// TIA Portal V16 export
// export: Created 2022-05-05T19:56:47.8854088Z, ExportSetting WithDefaults, DisplayName Totally Integrated Automation Portal, DisplayVersion V16 Update 2, DisplayName TIA Portal Version Control Interface, DisplayVersion V16 Update 2, DisplayName TIA Portal Openness, DisplayVersion V16 Update 2, DisplayName SINAMICS Startdrive Advanced, DisplayVersion V16 Update 5, DisplayName SINAMICS Startdrive G130, G150, S120, S150, SINAMICS MV, S210, DisplayVersion V16 Update 5, DisplayName SINAMICS Startdrive G110M, G120, G120C, G120D, G120P, G115D, DisplayVersion V16 Update 5, DisplayName STEP 7 Professional, DisplayVersion V16 Update 2, DisplayName SIMATIC Energy Suite, DisplayVersion V16, DisplayName STEP 7 Safety, DisplayVersion V16, DisplayName SINUMERIK 840D sl STEP 7 Toolbox, DisplayVersion V16, DisplayName Simocode ES, DisplayVersion V16, DisplayName WinCC Professional, DisplayVersion V16 Update 2, DisplayName SIMATIC Visualization Architect, DisplayVersion V16
ORGANIZATION_BLOCK "Main"   // OB1, LAD, ProgramCycle
TITLE = "Main Program Sweep (Cycle)"
{ S7_Optimized_Access := 'TRUE' }
VERSION : 0.1
// stored: AutoNumber true, IsIECCheckEnabled false, SetENOAutomatically false
   VAR_INPUT
      Initial_Call : Bool;   // Initial call of this OB
      Remanence : Bool;   // =True, if remanent data are available
   END_VAR
   VAR_TEMP   // added for the SCL form of the ladder/FBD networks
      _w1 : Bool;
      _w2 : Bool;
      _w3 : Bool;
      _w4 : Bool;
   END_VAR
BEGIN

REGION Network 1: Reset
   // Detect when Factory I/O starts running, reset state
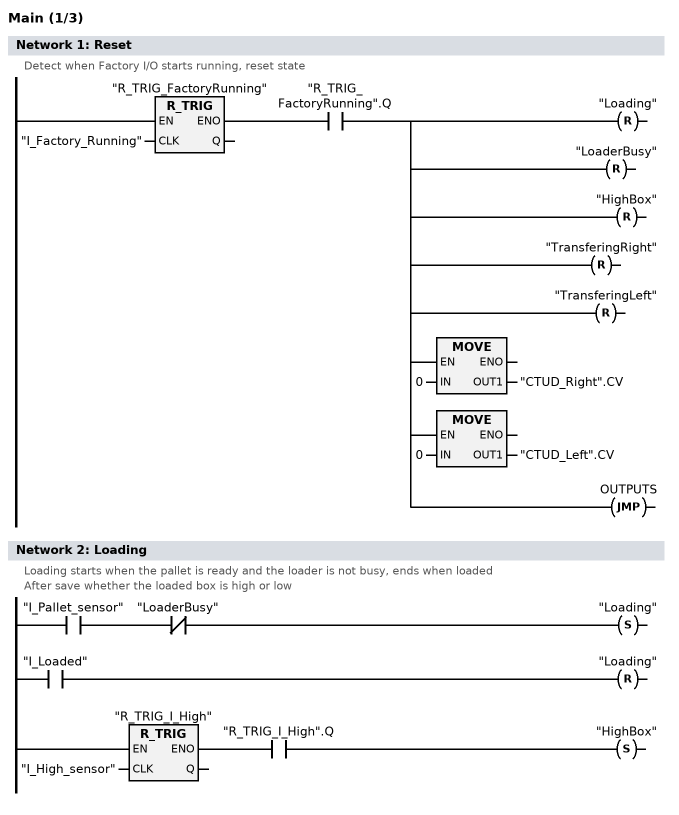
   RUNG wire#powerrail
      "R_TRIG_FactoryRunning".R_TRIG(CLK := "I_Factory_Running", Q =>)
      Contact( "R_TRIG_FactoryRunning".Q )
      wire#w1
      R_Coil( "Loading" )
   END_RUNG
   RUNG wire#w1
      R_Coil( "LoaderBusy" )
   END_RUNG
   RUNG wire#w1
      R_Coil( "HighBox" )
   END_RUNG
   RUNG wire#w1
      R_Coil( "TransferingRight" )
   END_RUNG
   RUNG wire#w1
      R_Coil( "TransferingLeft" )
   END_RUNG
   RUNG wire#w1
      Move(in := 0, out1 => "CTUD_Right".CV)
   END_RUNG
   RUNG wire#w1
      Move(in := 0, out1 => "CTUD_Left".CV)
   END_RUNG
   RUNG wire#w1
      JumpCoil( OUTPUTS )
   END_RUNG
   // the same network as SCL:
   "R_TRIG_FactoryRunning"(CLK := "I_Factory_Running", ENO => #_w1);   // R_TRIG
   #_w2 := #_w1 AND "R_TRIG_FactoryRunning".Q;
   IF #_w2 THEN
       "Loading" := FALSE;
       "LoaderBusy" := FALSE;
       "HighBox" := FALSE;
       "TransferingRight" := FALSE;
       "TransferingLeft" := FALSE;
       "CTUD_Right".CV := 0;
       "CTUD_Left".CV := 0;
       GOTO OUTPUTS;
   END_IF;
END_REGION

REGION Network 2: Loading
   // Loading starts when the pallet is ready and the loader is not busy, ends when loaded
   // After save whether the loaded box is high or low
   RUNG wire#powerrail
      Contact( "I_Pallet_sensor" )
      I_Contact( "LoaderBusy" )
      S_Coil( "Loading" )
   END_RUNG
   RUNG wire#powerrail
      Contact( "I_Loaded" )
      R_Coil( "Loading" )
   END_RUNG
   RUNG wire#powerrail
      "R_TRIG_I_High".R_TRIG(CLK := "I_High_sensor", Q =>)
      Contact( "R_TRIG_I_High".Q )
      S_Coil( "HighBox" )
   END_RUNG
   // the same network as SCL:
   IF "I_Pallet_sensor" AND NOT "LoaderBusy" THEN "Loading" := TRUE; END_IF;
   IF "I_Loaded" THEN "Loading" := FALSE; END_IF;
   "R_TRIG_I_High"(CLK := "I_High_sensor", ENO => #_w1);   // R_TRIG
   IF #_w1 AND "R_TRIG_I_High".Q THEN "HighBox" := TRUE; END_IF;
END_REGION

REGION Network 3: Transfer
   // Decide where to transfer after loading
   // Loader busy if loading or transfering
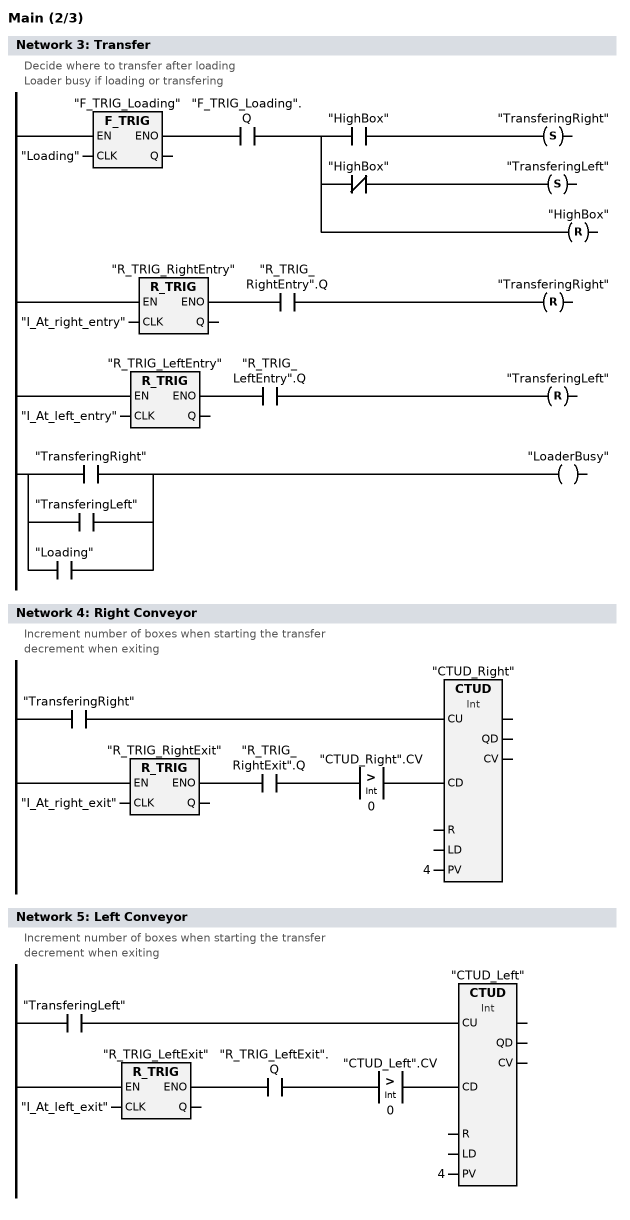
   RUNG wire#powerrail
      "F_TRIG_Loading".F_TRIG(CLK := "Loading", Q =>)
      Contact( "F_TRIG_Loading".Q )
      wire#w1
      Contact( "HighBox" )
      S_Coil( "TransferingRight" )
   END_RUNG
   RUNG wire#w1
      I_Contact( "HighBox" )
      S_Coil( "TransferingLeft" )
   END_RUNG
   RUNG wire#w1
      R_Coil( "HighBox" )
   END_RUNG
   RUNG wire#powerrail
      "R_TRIG_RightEntry".R_TRIG(CLK := "I_At_right_entry", Q =>)
      Contact( "R_TRIG_RightEntry".Q )
      R_Coil( "TransferingRight" )
   END_RUNG
   RUNG wire#powerrail
      "R_TRIG_LeftEntry".R_TRIG(CLK := "I_At_left_entry", Q =>)
      Contact( "R_TRIG_LeftEntry".Q )
      R_Coil( "TransferingLeft" )
   END_RUNG
   RUNG wire#powerrail
      Contact( "TransferingRight" )
      wire#w2
      Coil( "LoaderBusy" )
   END_RUNG
   RUNG wire#powerrail
      Contact( "TransferingLeft" )
   END_RUNG wire#w2
   RUNG wire#powerrail
      Contact( "Loading" )
   END_RUNG wire#w2
   // the same network as SCL:
   "F_TRIG_Loading"(CLK := "Loading", ENO => #_w1);   // F_TRIG
   #_w2 := #_w1 AND "F_TRIG_Loading".Q;
   IF #_w2 AND "HighBox" THEN "TransferingRight" := TRUE; END_IF;
   IF #_w2 AND NOT "HighBox" THEN "TransferingLeft" := TRUE; END_IF;
   IF #_w2 THEN "HighBox" := FALSE; END_IF;
   "R_TRIG_RightEntry"(CLK := "I_At_right_entry", ENO => #_w3);   // R_TRIG
   IF #_w3 AND "R_TRIG_RightEntry".Q THEN "TransferingRight" := FALSE; END_IF;
   "R_TRIG_LeftEntry"(CLK := "I_At_left_entry", ENO => #_w4);   // R_TRIG
   IF #_w4 AND "R_TRIG_LeftEntry".Q THEN "TransferingLeft" := FALSE; END_IF;
   "LoaderBusy" := "TransferingRight" OR "TransferingLeft" OR "Loading";
END_REGION

REGION Network 4: Right Conveyor
   // Increment number of boxes when starting the transfer
   // decrement when exiting
   RUNG wire#powerrail
      Contact( "TransferingRight" )
      { S7_Templates := "value_type := Int" } "CTUD_Right".CTUD(cd := wire#w1, r :=, ld :=, pv := 4, qd =>, cv =>)
   END_RUNG
   RUNG wire#powerrail
      "R_TRIG_RightExit".R_TRIG(CLK := "I_At_right_exit", Q =>)
      Contact( "R_TRIG_RightExit".Q )
      { S7_Templates := "SrcType := Int" } GT_Contact(in1 := "CTUD_Right".CV, in2 := 0)
   END_RUNG wire#w1
   // the same network as SCL:
   "R_TRIG_RightExit"(CLK := "I_At_right_exit", ENO => #_w1);   // R_TRIG
   "CTUD_Right".CTUD(CU := "TransferingRight",
                     CD := #_w1 AND "R_TRIG_RightExit".Q AND ("CTUD_Right".CV > 0),
                     PV := 4);
END_REGION

REGION Network 5: Left Conveyor
   // Increment number of boxes when starting the transfer
   // decrement when exiting
   RUNG wire#powerrail
      Contact( "TransferingLeft" )
      { S7_Templates := "value_type := Int" } "CTUD_Left".CTUD(cd := wire#w1, r :=, ld :=, pv := 4, qd =>, cv =>)
   END_RUNG
   RUNG wire#powerrail
      "R_TRIG_LeftExit".R_TRIG(CLK := "I_At_left_exit", Q =>)
      Contact( "R_TRIG_LeftExit".Q )
      { S7_Templates := "SrcType := Int" } GT_Contact(in1 := "CTUD_Left".CV, in2 := 0)
   END_RUNG wire#w1
   // the same network as SCL:
   "R_TRIG_LeftExit"(CLK := "I_At_left_exit", ENO => #_w1);   // R_TRIG
   "CTUD_Left".CTUD(CU := "TransferingLeft",
                    CD := #_w1 AND "R_TRIG_LeftExit".Q AND ("CTUD_Left".CV > 0),
                    PV := 4);
END_REGION

REGION Network 6: Set the outputs
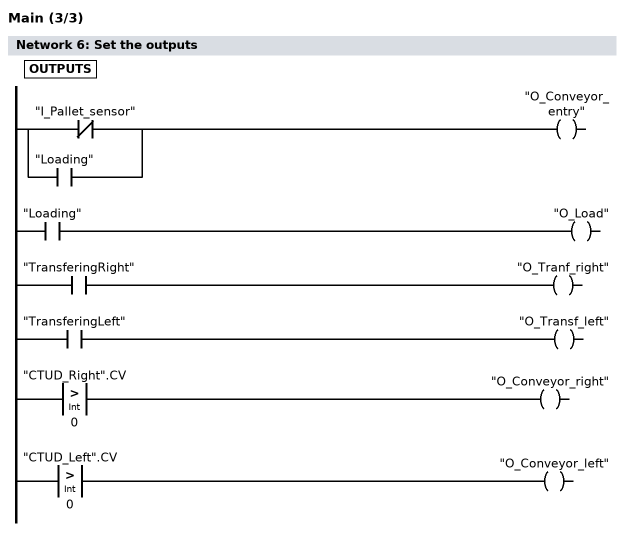
   Label( OUTPUTS )
   RUNG wire#powerrail
      I_Contact( "I_Pallet_sensor" )
      wire#w1
      Coil( "O_Conveyor_entry" )
   END_RUNG
   RUNG wire#powerrail
      Contact( "Loading" )
   END_RUNG wire#w1
   RUNG wire#powerrail
      Contact( "Loading" )
      Coil( "O_Load" )
   END_RUNG
   RUNG wire#powerrail
      Contact( "TransferingRight" )
      Coil( "O_Tranf_right" )
   END_RUNG
   RUNG wire#powerrail
      Contact( "TransferingLeft" )
      Coil( "O_Transf_left" )
   END_RUNG
   RUNG wire#powerrail
      { S7_Templates := "SrcType := Int" } GT_Contact(in1 := "CTUD_Right".CV, in2 := 0)
      Coil( "O_Conveyor_right" )
   END_RUNG
   RUNG wire#powerrail
      { S7_Templates := "SrcType := Int" } GT_Contact(in1 := "CTUD_Left".CV, in2 := 0)
      Coil( "O_Conveyor_left" )
   END_RUNG
   // the same network as SCL:
   OUTPUTS:
   "O_Conveyor_entry" := NOT "I_Pallet_sensor" OR "Loading";
   "O_Load" := "Loading";
   "O_Tranf_right" := "TransferingRight";
   "O_Transf_left" := "TransferingLeft";
   "O_Conveyor_right" := "CTUD_Right".CV > 0;
   "O_Conveyor_left" := "CTUD_Left".CV > 0;
END_REGION
END_ORGANIZATION_BLOCK
